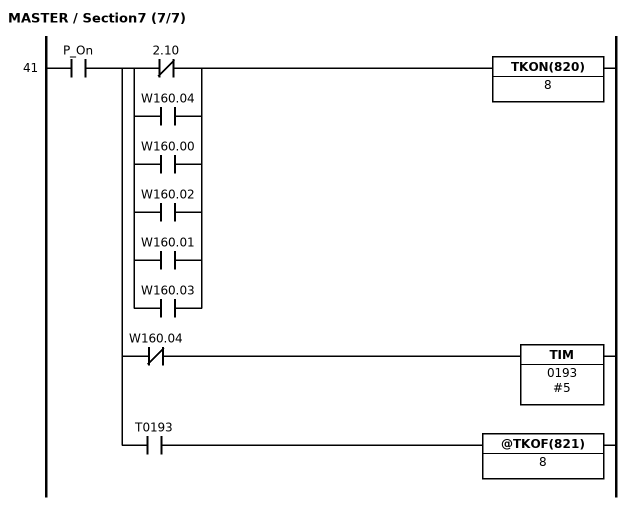
; [picture p24: MASTER / Section7, rungs 41-41]
; rung 41
LD P_On
OUT TR0
LDNOT 2.10
OR W160.04
OR W160.00
OR W160.02
OR W160.01
OR W160.03
ANDLD
TKON(820) 8
LD TR0
ANDNOT W160.04
TIM 0193 #5
LD TR0
AND T0193
@TKOF(821) 8  // 

### Section Section8

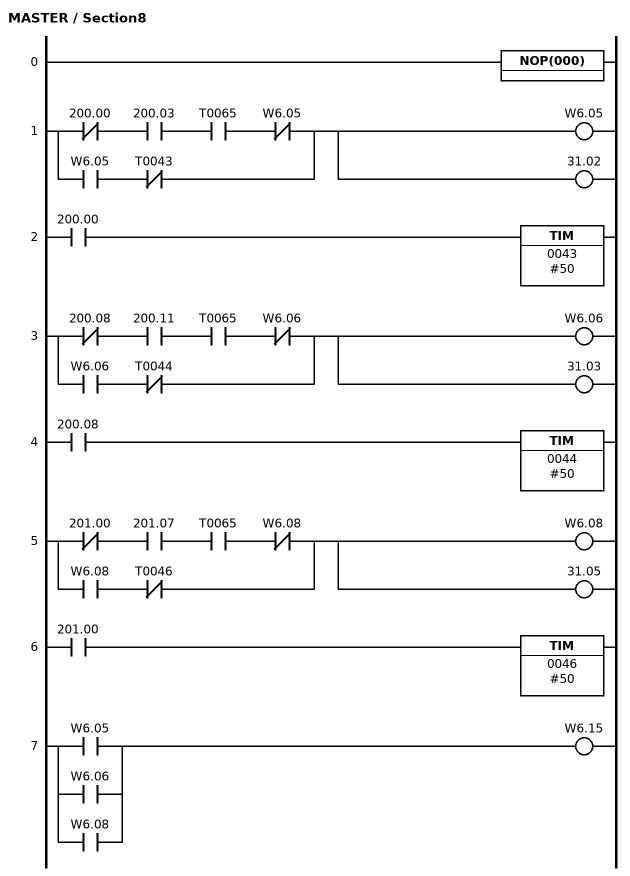
; rung 0
NOP(000)
; rung 1
// R
LDNOT 200.00
AND 200.03
AND T0065
ANDNOT W6.05
LD W6.05
ANDNOT T0043
ORLD
OUT W6.05
OUT 31.02
; rung 2
LD 200.00
TIM 0043 #50
; rung 3
// R
LDNOT 200.08
AND 200.11
AND T0065
ANDNOT W6.06
LD W6.06
ANDNOT T0044
ORLD
OUT W6.06
OUT 31.03
; rung 4
LD 200.08
TIM 0044 #50
; rung 5
// R
LDNOT 201.00
AND 201.07
AND T0065
ANDNOT W6.08
LD W6.08
ANDNOT T0046
ORLD
OUT W6.08
OUT 31.05
; rung 6
LD 201.00
TIM 0046 #50
; rung 7
// R
LD W6.05
OR W6.06
OR W6.08
OUT W6.15

### Section Section9

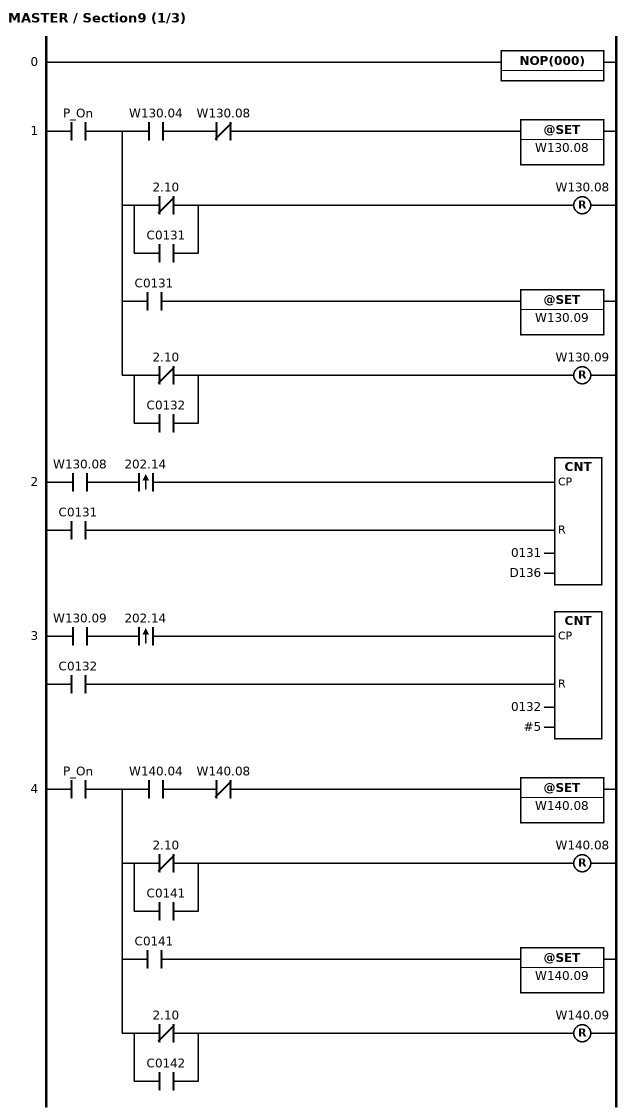
; rung 0
NOP(000)
; rung 1
LD P_On
OUT TR0
AND W130.04
ANDNOT W130.08
@SET W130.08
LD TR0
LDNOT 2.10
OR C0131
ANDLD
RSET W130.08
LD TR0
AND C0131
@SET W130.09
LD TR0
LDNOT 2.10
OR C0132
ANDLD
RSET W130.09
; rung 2
LD W130.08
@AND 202.14
LD C0131
CNT 0131 D136
; rung 3
LD W130.09
@AND 202.14
LD C0132
CNT 0132 #5
; rung 4
LD P_On
OUT TR0
AND W140.04
ANDNOT W140.08
@SET W140.08
LD TR0
LDNOT 2.10
OR C0141
ANDLD
RSET W140.08
LD TR0
AND C0141
@SET W140.09
LD TR0
LDNOT 2.10
OR C0142
ANDLD
RSET W140.09

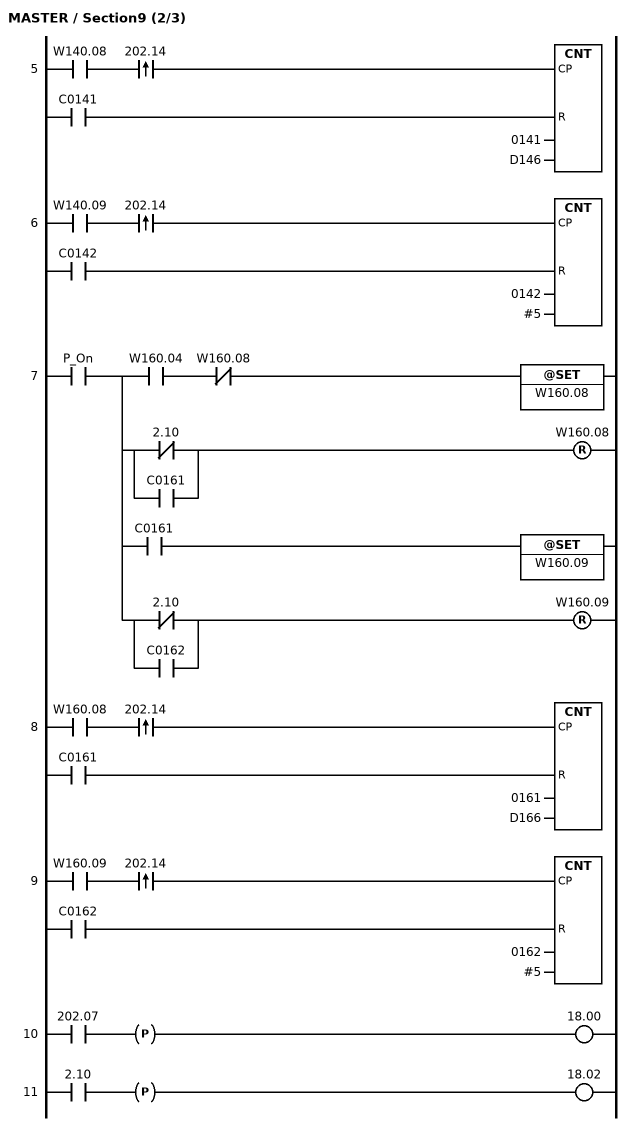
; rung 5
LD W140.08
@AND 202.14
LD C0141
CNT 0141 D146
; rung 6
LD W140.09
@AND 202.14
LD C0142
CNT 0142 #5
; rung 7
LD P_On
OUT TR0
AND W160.04
ANDNOT W160.08
@SET W160.08
LD TR0
LDNOT 2.10
OR C0161
ANDLD
RSET W160.08
LD TR0
AND C0161
@SET W160.09
LD TR0
LDNOT 2.10
OR C0162
ANDLD
RSET W160.09
; rung 8
LD W160.08
@AND 202.14
LD C0161
CNT 0161 D166
; rung 9
LD W160.09
@AND 202.14
LD C0162
CNT 0162 #5
; rung 10
LD 202.07
UP(521)
OUT 18.00
; rung 11
LD 2.10
UP(521)
OUT 18.02

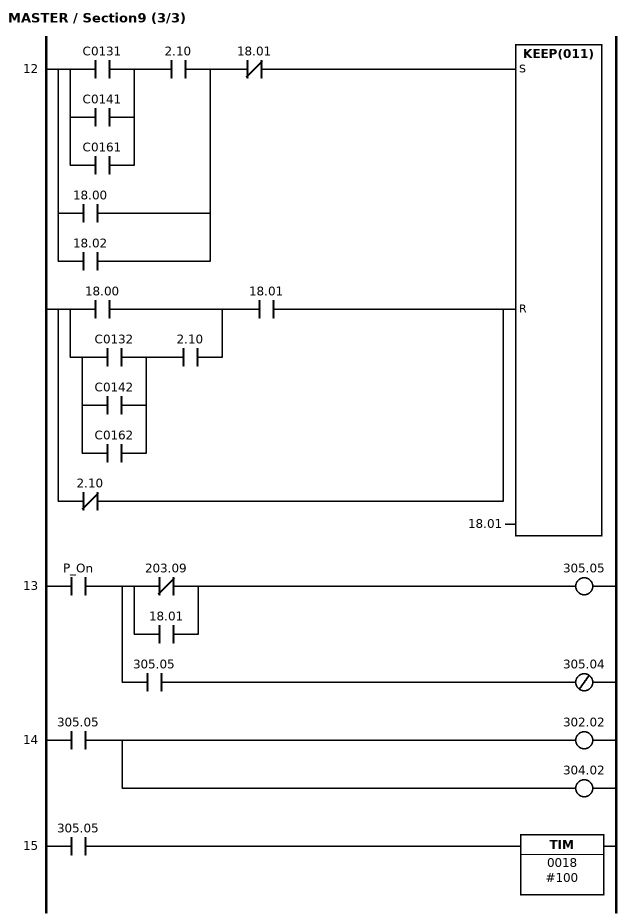
; rung 12
// R
LD C0131
OR C0141
OR C0161
AND 2.10
OR 18.00
OR 18.02
ANDNOT 18.01
LD 18.00
LD C0132
OR C0142
OR C0162
AND 2.10
ORLD
AND 18.01
ORNOT 2.10
KEEP(011) 18.01
; rung 13
LD P_On
OUT TR0
LDNOT 203.09
OR 18.01
ANDLD
OUT 305.05
LD TR0
AND 305.05
OUTNOT 305.04
; rung 14
LD 305.05
OUT 302.02
OUT 304.02
; rung 15
LD 305.05
TIM 0018 #100

### Section Section10

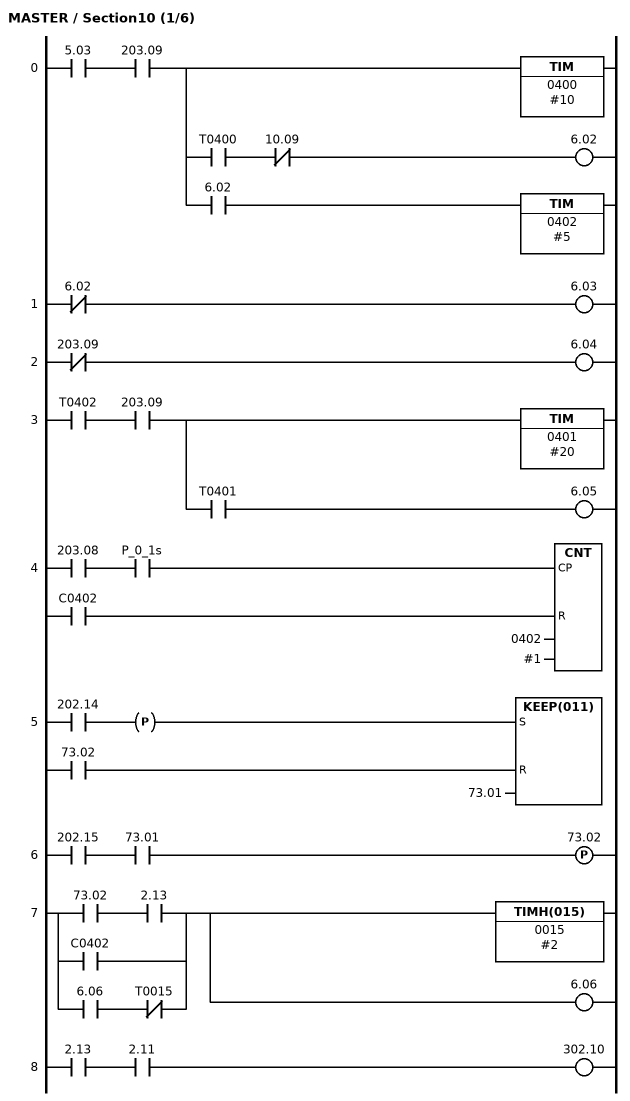
; rung 0
// R
LD 5.03
AND 203.09
OUT TR0
TIM 0400 #10
AND T0400
ANDNOT 10.09
OUT 6.02
LD TR0
AND 6.02
TIM 0402 #5
; rung 1
LDNOT 6.02
OUT 6.03
; rung 2
LDNOT 203.09
OUT 6.04
; rung 3
LD T0402
AND 203.09
TIM 0401 #20
AND T0401
OUT 6.05
; rung 4
LD 203.08
AND P_0_1s
LD C0402
CNT 0402 #1
; rung 5
LD 202.14
UP(521)
LD 73.02
KEEP(011) 73.01
; rung 6
LD 202.15
AND 73.01
DIFU(013) 73.02
; rung 7
LD 73.02
AND 2.13
OR C0402
LD 6.06
ANDNOT T0015
ORLD
TIMH(015) 0015 #2
OUT 6.06
; rung 8
LD 2.13
AND 2.11
OUT 302.10

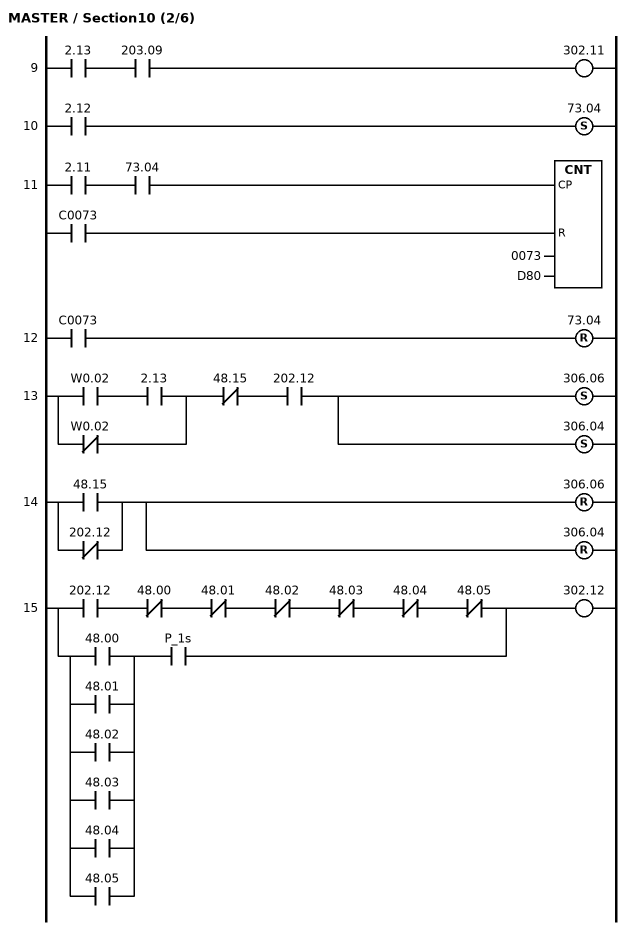
; rung 9
LD 2.13
AND 203.09
OUT 302.11
; rung 10
LD 2.12
SET 73.04
; rung 11
LD 2.11
AND 73.04
LD C0073
CNT 0073 D80
; rung 12
LD C0073
RSET 73.04
; rung 13
LD W0.02
AND 2.13
ORNOT W0.02
ANDNOT 48.15
AND 202.12
SET 306.06
SET 306.04
; rung 14
LD 48.15
ORNOT 202.12
RSET 306.06
RSET 306.04
; rung 15
LD 202.12
ANDNOT 48.00
ANDNOT 48.01
ANDNOT 48.02
ANDNOT 48.03
ANDNOT 48.04
ANDNOT 48.05
LD 48.00
OR 48.01
OR 48.02
OR 48.03
OR 48.04
OR 48.05
AND P_1s
ORLD
OUT 302.12

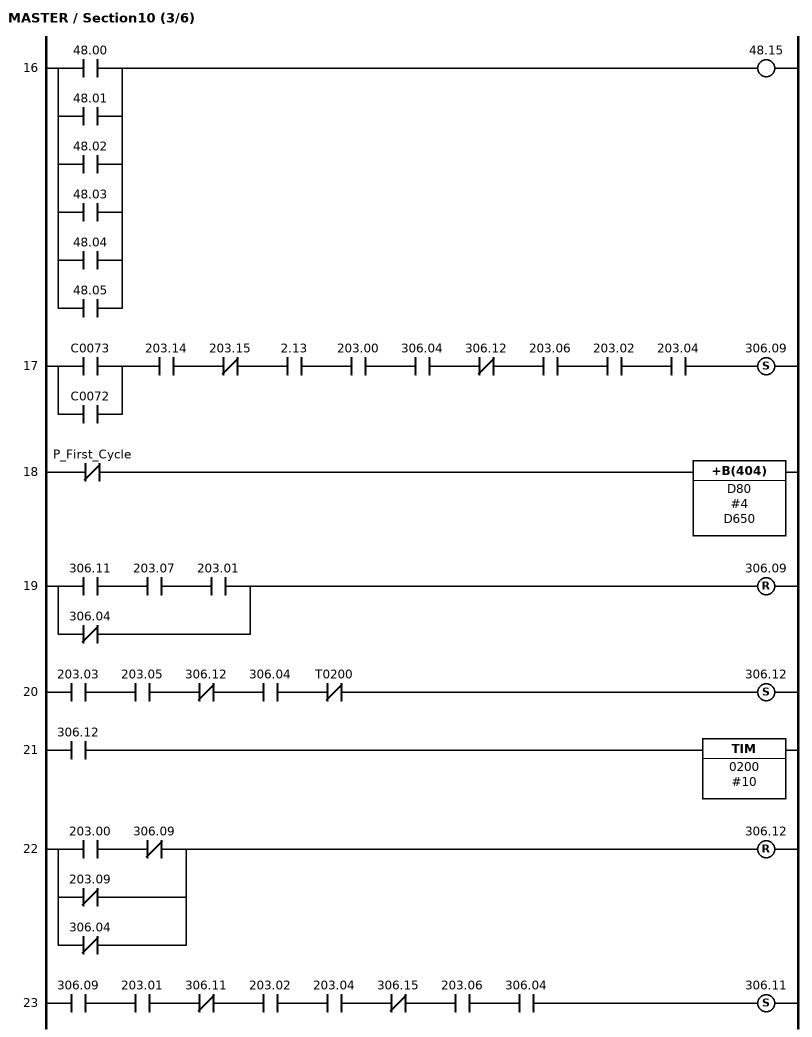
; rung 16
LD 48.00
OR 48.01
OR 48.02
OR 48.03
OR 48.04
OR 48.05
OUT 48.15
; rung 17
// R
LD C0073
OR C0072
AND 203.14
ANDNOT 203.15
AND 2.13
AND 203.00
AND 306.04
ANDNOT 306.12
AND 203.06
AND 203.02
AND 203.04
SET 306.09
; rung 18
LDNOT P_First_Cycle
+B(404) D80 #4 D650
; rung 19
LD 306.11
AND 203.07
AND 203.01
ORNOT 306.04
RSET 306.09
; rung 20
LD 203.03
AND 203.05
ANDNOT 306.12
AND 306.04
ANDNOT T0200
SET 306.12
; rung 21
LD 306.12
TIM 0200 #10
; rung 22
LD 203.00
ANDNOT 306.09
ORNOT 203.09
ORNOT 306.04
RSET 306.12
; rung 23
LD 306.09
AND 203.01
ANDNOT 306.11
AND 203.02
AND 203.04
ANDNOT 306.15
AND 203.06
AND 306.04
SET 306.11

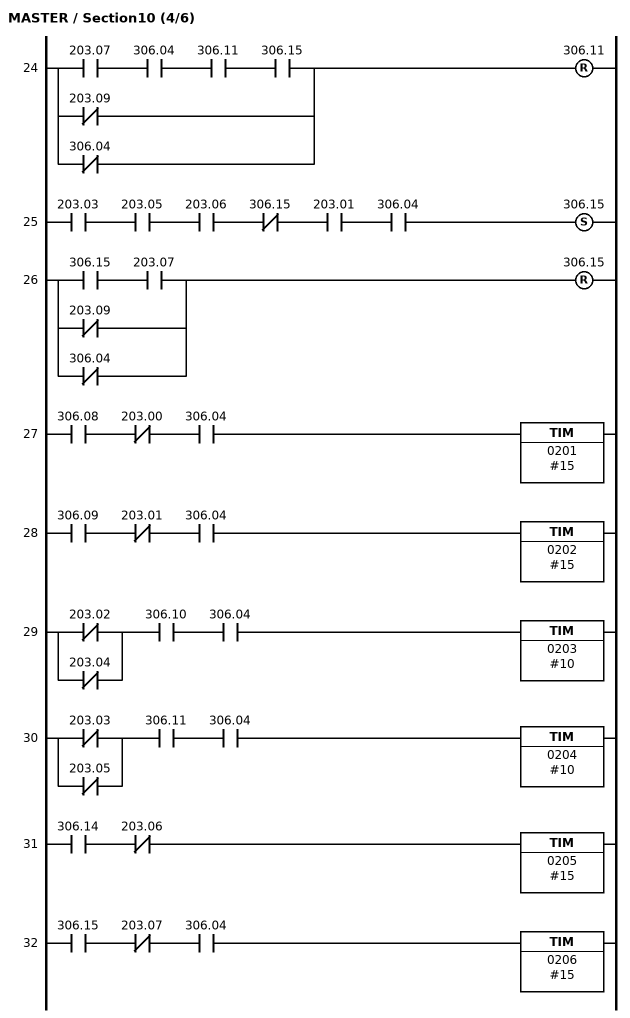
; rung 24
LD 203.07
AND 306.04
AND 306.11
AND 306.15
ORNOT 203.09
ORNOT 306.04
RSET 306.11
; rung 25
LD 203.03
AND 203.05
AND 203.06
ANDNOT 306.15
AND 203.01
AND 306.04
SET 306.15
; rung 26
LD 306.15
AND 203.07
ORNOT 203.09
ORNOT 306.04
RSET 306.15
; rung 27
LD 306.08
ANDNOT 203.00
AND 306.04
TIM 0201 #15
; rung 28
LD 306.09
ANDNOT 203.01
AND 306.04
TIM 0202 #15
; rung 29
LDNOT 203.02
ORNOT 203.04
AND 306.10
AND 306.04
TIM 0203 #10
; rung 30
LDNOT 203.03
ORNOT 203.05
AND 306.11
AND 306.04
TIM 0204 #10
; rung 31
LD 306.14
ANDNOT 203.06
TIM 0205 #15
; rung 32
LD 306.15
ANDNOT 203.07
AND 306.04
TIM 0206 #15

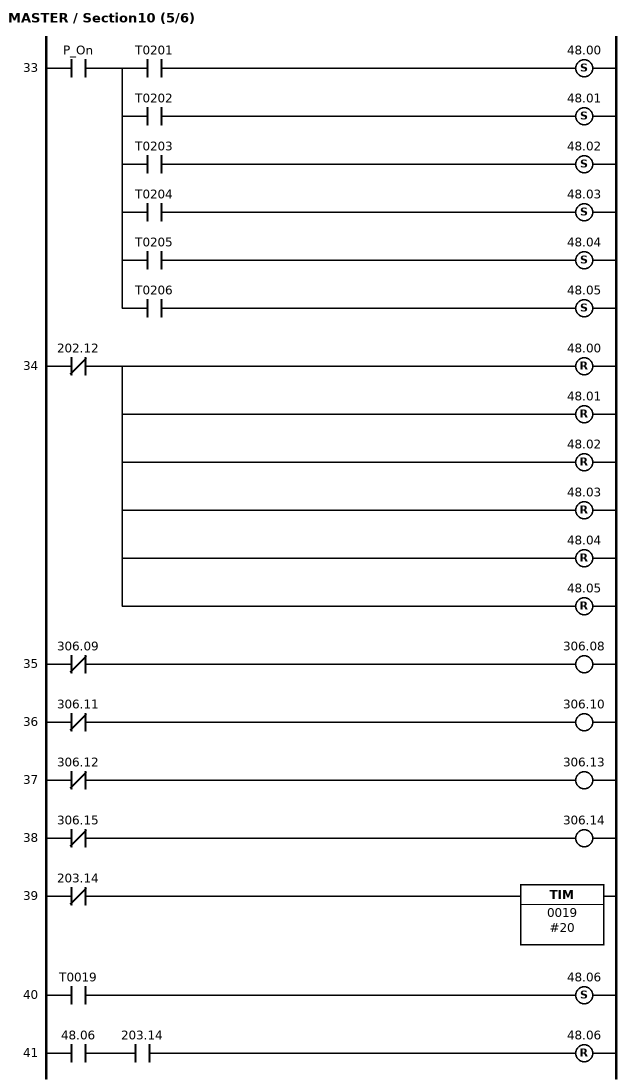
; rung 33
LD P_On
OUT TR0
AND T0201
SET 48.00
LD TR0
AND T0202
SET 48.01
LD TR0
AND T0203
SET 48.02
LD TR0
AND T0204
SET 48.03
LD TR0
AND T0205
SET 48.04
LD TR0
AND T0206
SET 48.05
; rung 34
LDNOT 202.12
RSET 48.00
RSET 48.01
RSET 48.02
RSET 48.03
RSET 48.04
RSET 48.05
; rung 35
LDNOT 306.09
OUT 306.08
; rung 36
LDNOT 306.11
OUT 306.10
; rung 37
LDNOT 306.12
OUT 306.13
; rung 38
LDNOT 306.15
OUT 306.14
; rung 39
// R
LDNOT 203.14
TIM 0019 #20
; rung 40
LD T0019
SET 48.06
; rung 41
LD 48.06
AND 203.14
RSET 48.06

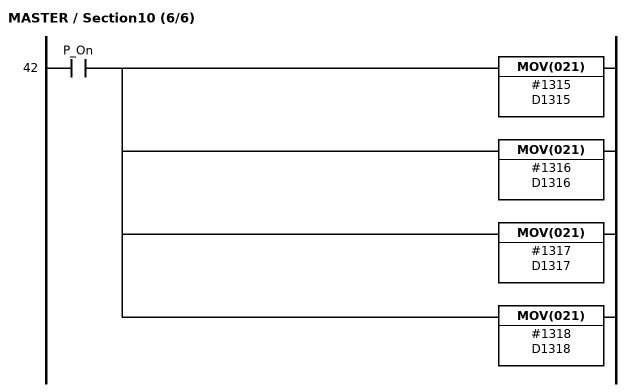
; rung 42
LD P_On
MOV(021) #1315 D1315
MOV(021) #1316 D1316
MOV(021) #1317 D1317
MOV(021) #1318 D1318

### Section Section11

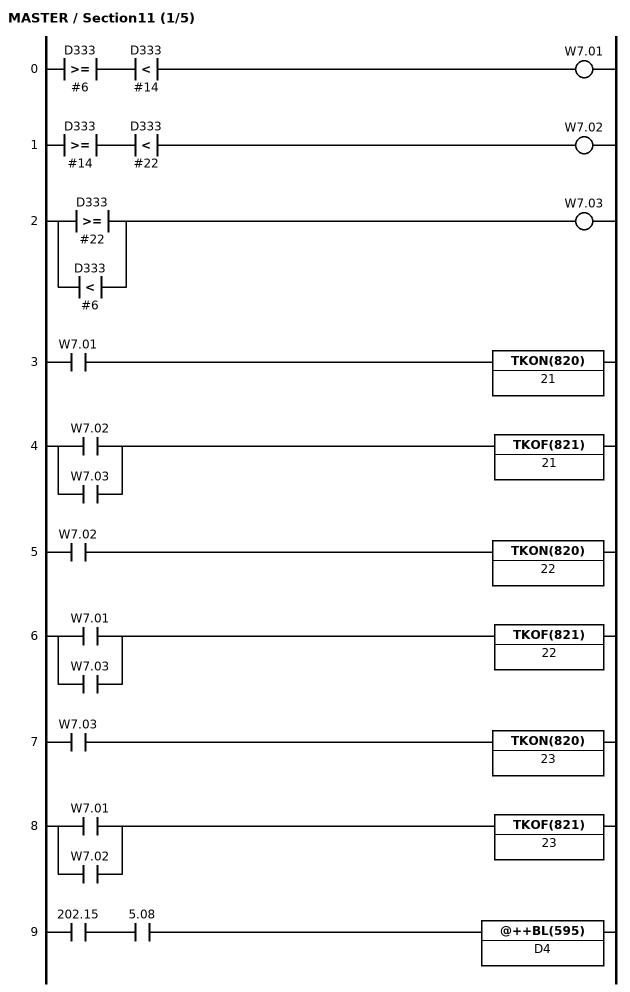
; rung 0
// R
LD>=(325) D333 #6
AND<(310) D333 #14
OUT W7.01  // 
; rung 1
LD>=(325) D333 #14
AND<(310) D333 #22
OUT W7.02  // 
; rung 2
LD>=(325) D333 #22
OR<(310) D333 #6
OUT W7.03  // 
; rung 3
LD W7.01
TKON(820) 21
; rung 4
LD W7.02
OR W7.03
TKOF(821) 21
; rung 5
LD W7.02
TKON(820) 22
; rung 6
LD W7.01
OR W7.03
TKOF(821) 22
; rung 7
LD W7.03
TKON(820) 23
; rung 8
LD W7.01
OR W7.02
TKOF(821) 23
; rung 9
LD 202.15
AND 5.08
@++BL(595) D4  // 

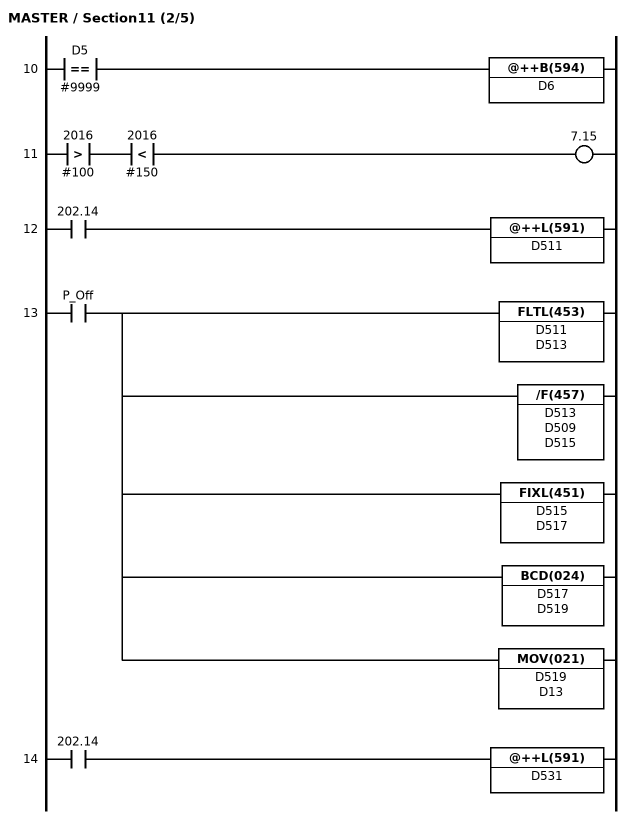
; rung 10
LD=(300) D5 #9999
@++B(594) D6
; rung 11
LD>(320) 2016 #100
AND<(310) 2016 #150
OUT 7.15
; rung 12
// R
LD 202.14
@++L(591) D511  // 
; rung 13
// R
LD P_Off
FLTL(453) D511 D513
/F(457) D513 D509 D515
FIXL(451) D515 D517
BCD(024) D517 D519
MOV(021) D519 D13
; rung 14
// R
LD 202.14
@++L(591) D531  // 

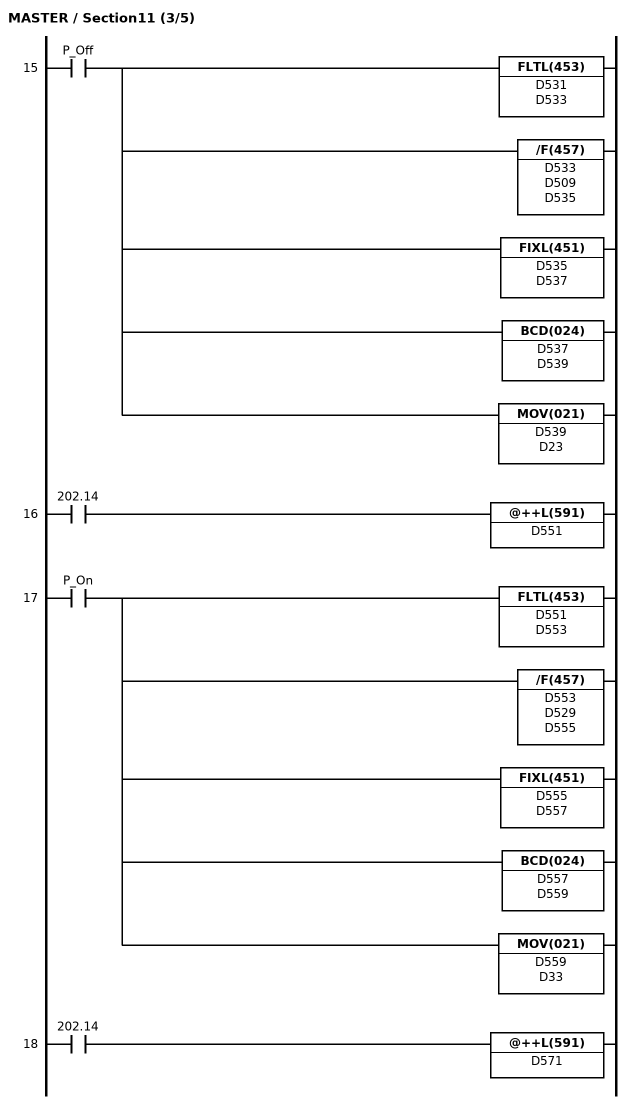
; rung 15
LD P_Off
FLTL(453) D531 D533
/F(457) D533 D509 D535
FIXL(451) D535 D537
BCD(024) D537 D539
MOV(021) D539 D23
; rung 16
// R
LD 202.14
@++L(591) D551  // 
; rung 17
LD P_On
FLTL(453) D551 D553
/F(457) D553 D529 D555
FIXL(451) D555 D557
BCD(024) D557 D559
MOV(021) D559 D33
; rung 18
// R
LD 202.14
@++L(591) D571  // 

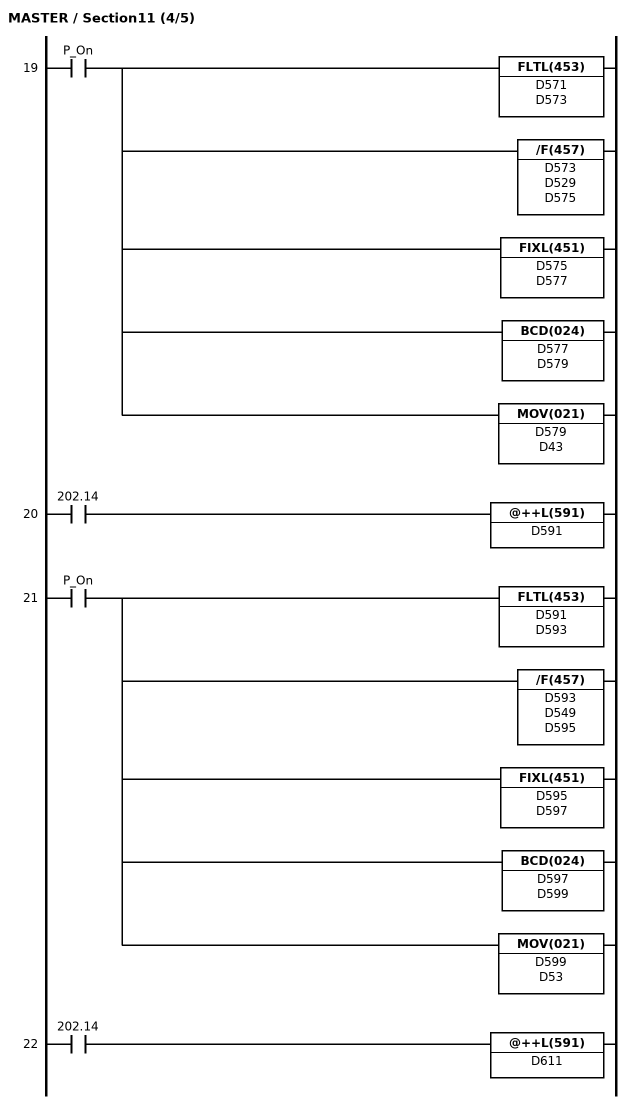
; rung 19
LD P_On
FLTL(453) D571 D573
/F(457) D573 D529 D575
FIXL(451) D575 D577
BCD(024) D577 D579
MOV(021) D579 D43
; rung 20
// R
LD 202.14
@++L(591) D591  // 
; rung 21
LD P_On
FLTL(453) D591 D593
/F(457) D593 D549 D595
FIXL(451) D595 D597
BCD(024) D597 D599
MOV(021) D599 D53
; rung 22
// R
LD 202.14
@++L(591) D611  // 

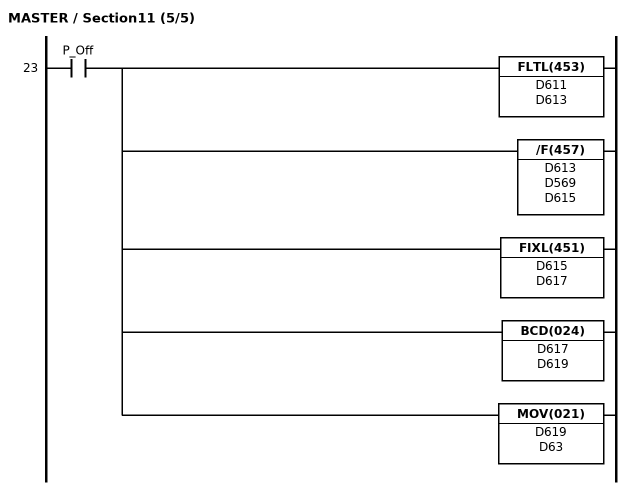
; rung 23
LD P_Off
FLTL(453) D611 D613
/F(457) D613 D569 D615
FIXL(451) D615 D617
BCD(024) D617 D619
MOV(021) D619 D63

### Section Section12

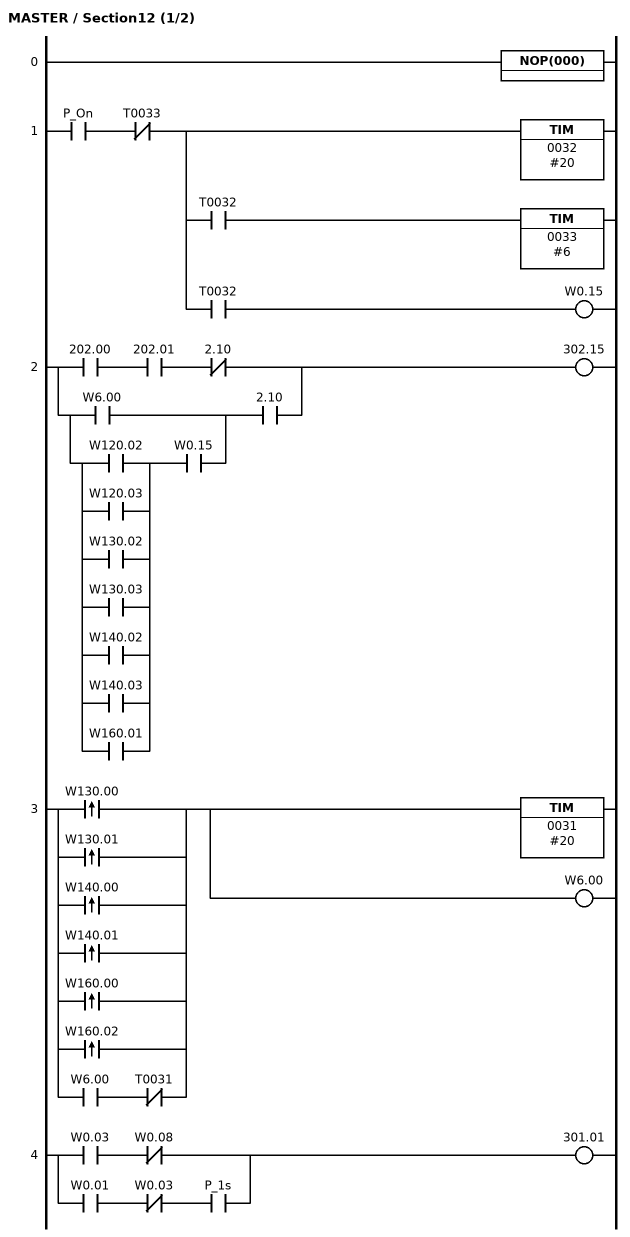
; rung 0
NOP(000)
; rung 1
LD P_On
ANDNOT T0033
OUT TR0
TIM 0032 #20
AND T0032
TIM 0033 #6
LD TR0
AND T0032
OUT W0.15
; rung 2
// R
LD 202.00
AND 202.01
ANDNOT 2.10
LD W6.00
LD W120.02
OR W120.03
OR W130.02
OR W130.03
OR W140.02
OR W140.03
OR W160.01
AND W0.15
ORLD
AND 2.10
ORLD
OUT 302.15
; rung 3
// R
@LD W130.00
@OR W130.01
@OR W140.00
@OR W140.01
@OR W160.00
@OR W160.02
LD W6.00
ANDNOT T0031
ORLD
TIM 0031 #20
OUT W6.00
; rung 4
// R
LD W0.03
ANDNOT W0.08
LD W0.01
ANDNOT W0.03
AND P_1s
ORLD
OUT 301.01

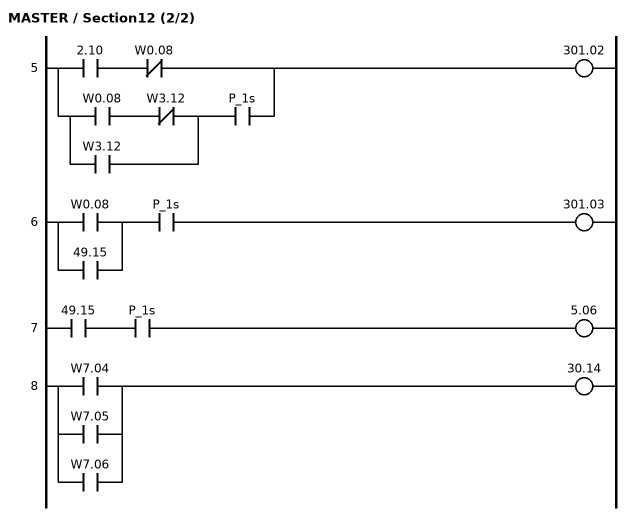
; rung 5
// R
LD 2.10
ANDNOT W0.08
LD W0.08
ANDNOT W3.12
OR W3.12
AND P_1s
ORLD
OUT 301.02
; rung 6
// R
LD W0.08
OR 49.15
AND P_1s
OUT 301.03
; rung 7
LD 49.15
AND P_1s
OUT 5.06
; rung 8
// R
LD W7.04
OR W7.05
OR W7.06
OUT 30.14

### Section Section13

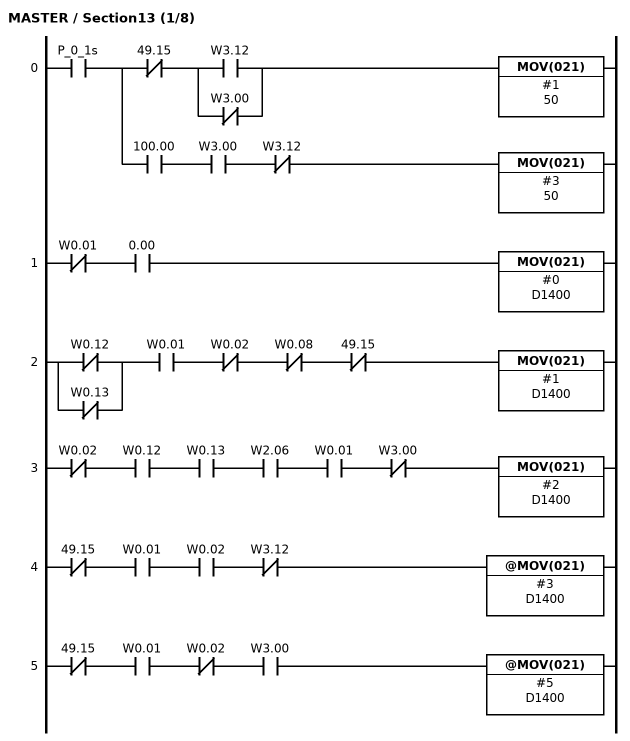
; rung 0
// R
LD P_0_1s
OUT TR0
ANDNOT 49.15
LD W3.12
ORNOT W3.00
ANDLD
MOV(021) #1 50
LD TR0
AND 100.00
AND W3.00
ANDNOT W3.12
MOV(021) #3 50
; rung 1
LDNOT W0.01
AND 0.00
MOV(021) #0 D1400
; rung 2
LDNOT W0.12
ORNOT W0.13
AND W0.01
ANDNOT W0.02
ANDNOT W0.08
ANDNOT 49.15
MOV(021) #1 D1400
; rung 3
LDNOT W0.02
AND W0.12
AND W0.13
AND W2.06
AND W0.01
ANDNOT W3.00
MOV(021) #2 D1400
; rung 4
LDNOT 49.15
AND W0.01
AND W0.02
ANDNOT W3.12
@MOV(021) #3 D1400
; rung 5
LDNOT 49.15
AND W0.01
ANDNOT W0.02
AND W3.00
@MOV(021) #5 D1400

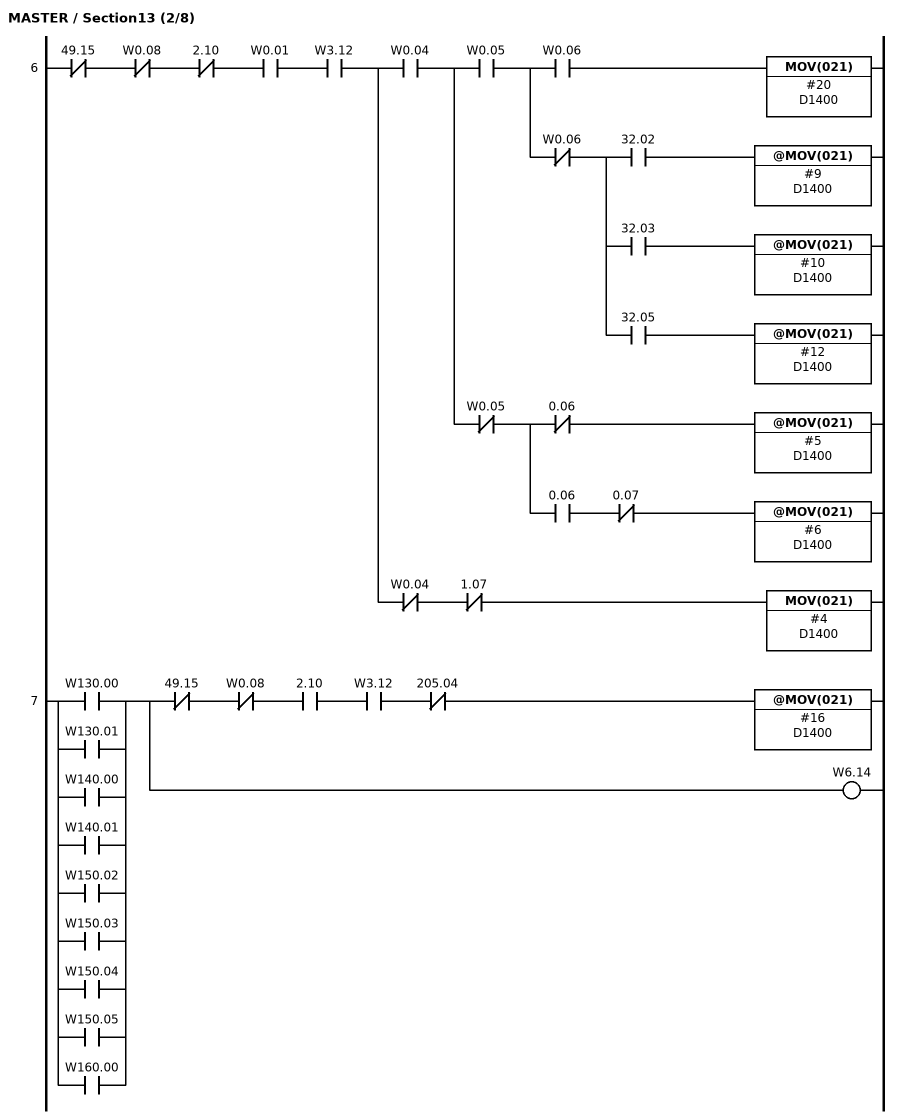
; rung 6
LDNOT 49.15
ANDNOT W0.08
ANDNOT 2.10
AND W0.01
AND W3.12
OUT TR0
AND W0.04
OUT TR1
AND W0.05
OUT TR2
AND W0.06
MOV(021) #20 D1400
LD TR2
ANDNOT W0.06
OUT TR2
AND 32.02
@MOV(021) #9 D1400
LD TR2
AND 32.03
@MOV(021) #10 D1400
LD TR2
AND 32.05
@MOV(021) #12 D1400
LD TR1
ANDNOT W0.05
OUT TR1
ANDNOT 0.06
@MOV(021) #5 D1400
LD TR1
AND 0.06
ANDNOT 0.07
@MOV(021) #6 D1400
LD TR0
ANDNOT W0.04
ANDNOT 1.07
MOV(021) #4 D1400
; rung 7
LD W130.00
OR W130.01
OR W140.00
OR W140.01
OR W150.02
OR W150.03
OR W150.04
OR W150.05
OR W160.00
OUT TR0
ANDNOT 49.15
ANDNOT W0.08
AND 2.10
AND W3.12
ANDNOT 205.04
@MOV(021) #16 D1400
LD TR0
OUT W6.14

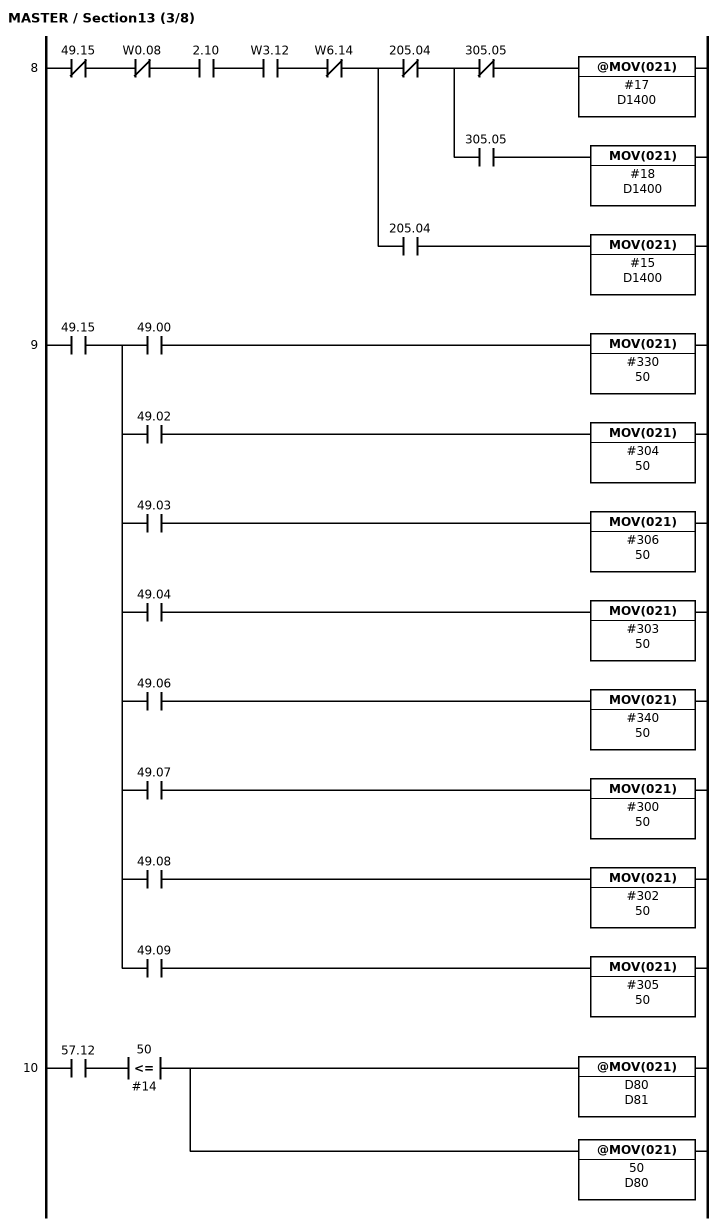
; rung 8
LDNOT 49.15
ANDNOT W0.08
AND 2.10
AND W3.12
ANDNOT W6.14
OUT TR0
ANDNOT 205.04
OUT TR1
ANDNOT 305.05
@MOV(021) #17 D1400
LD TR1
AND 305.05
MOV(021) #18 D1400
LD TR0
AND 205.04
MOV(021) #15 D1400
; rung 9
LD 49.15
OUT TR0
AND 49.00
MOV(021) #330 50
LD TR0
AND 49.02
MOV(021) #304 50
LD TR0
AND 49.03
MOV(021) #306 50
LD TR0
AND 49.04
MOV(021) #303 50
LD TR0
AND 49.06
MOV(021) #340 50
LD TR0
AND 49.07
MOV(021) #300 50
LD TR0
AND 49.08
MOV(021) #302 50
LD TR0
AND 49.09
MOV(021) #305 50
; rung 10
// R
LD 57.12
AND<=(315) 50 #14
@MOV(021) D80 D81
@MOV(021) 50 D80

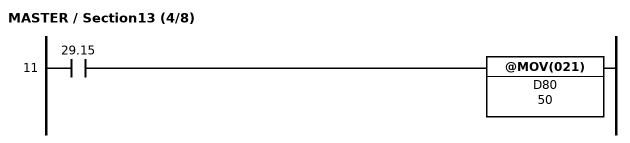
; rung 11
LD 29.15
@MOV(021) D80 50

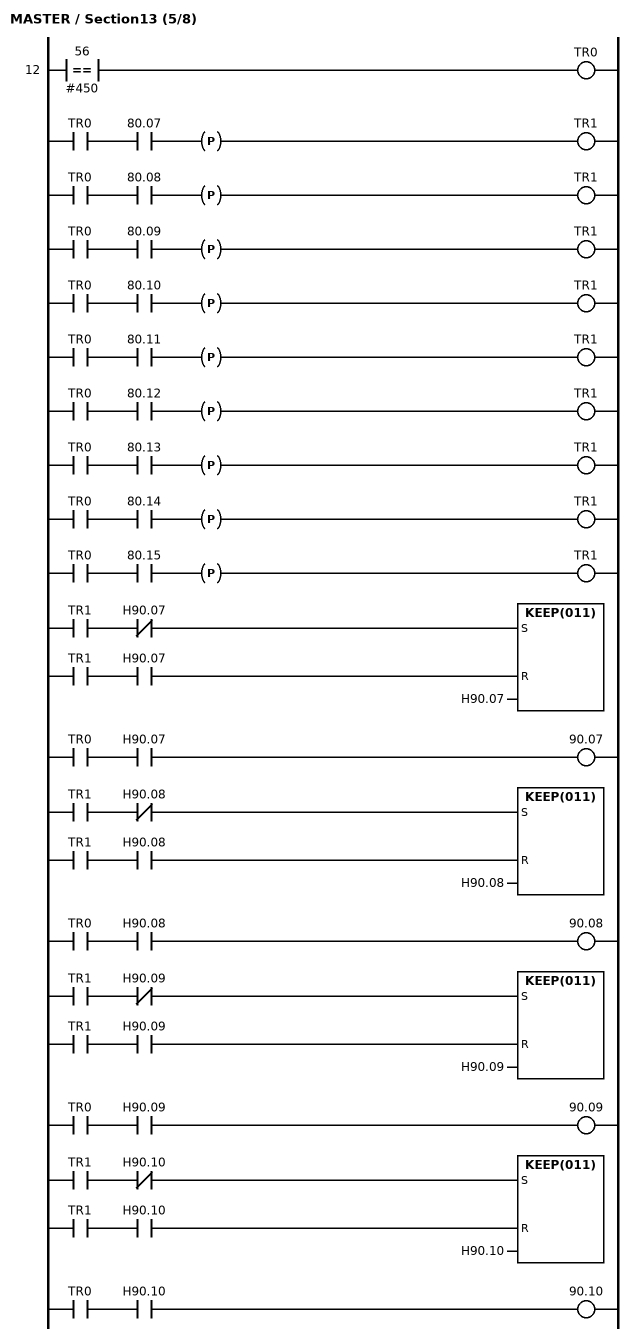

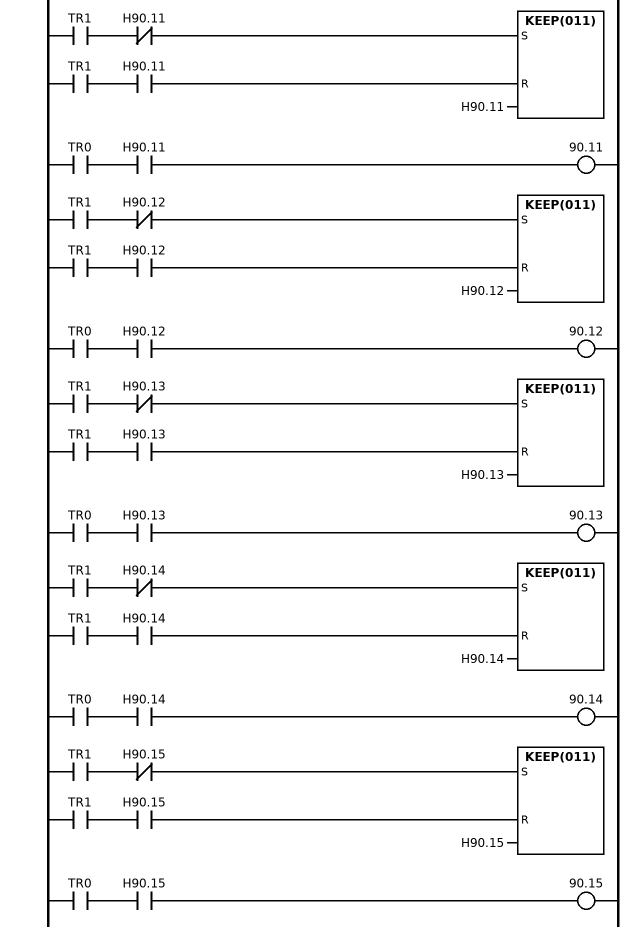
; rung 12
LD=(300) 56 #450
OUT TR0
AND 80.07
UP(521)
OUT TR1
ANDNOT H90.07
LD TR1
AND H90.07
KEEP(011) H90.07
LD TR0
AND H90.07
OUT 90.07
LD TR0
AND 80.08
UP(521)
OUT TR1
ANDNOT H90.08
LD TR1
AND H90.08
KEEP(011) H90.08
LD TR0
AND H90.08
OUT 90.08
LD TR0
AND 80.09
UP(521)
OUT TR1
ANDNOT H90.09
LD TR1
AND H90.09
KEEP(011) H90.09
LD TR0
AND H90.09
OUT 90.09
LD TR0
AND 80.10
UP(521)
OUT TR1
ANDNOT H90.10
LD TR1
AND H90.10
KEEP(011) H90.10
LD TR0
AND H90.10
OUT 90.10
LD TR0
AND 80.11
UP(521)
OUT TR1
ANDNOT H90.11
LD TR1
AND H90.11
KEEP(011) H90.11
LD TR0
AND H90.11
OUT 90.11
LD TR0
AND 80.12
UP(521)
OUT TR1
ANDNOT H90.12
LD TR1
AND H90.12
KEEP(011) H90.12
LD TR0
AND H90.12
OUT 90.12
LD TR0
AND 80.13
UP(521)
OUT TR1
ANDNOT H90.13
LD TR1
AND H90.13
KEEP(011) H90.13
LD TR0
AND H90.13
OUT 90.13
LD TR0
AND 80.14
UP(521)
OUT TR1
ANDNOT H90.14
LD TR1
AND H90.14
KEEP(011) H90.14
LD TR0
AND H90.14
OUT 90.14
LD TR0
AND 80.15
UP(521)
OUT TR1
ANDNOT H90.15
LD TR1
AND H90.15
KEEP(011) H90.15
LD TR0
AND H90.15
OUT 90.15

